PROGRAM main
  VAR
    SYSTEM_ON : BOOL := FALSE;
    SYS_READY : BOOL := FALSE;
    START_MEASURE : BOOL := FALSE;
    PZEM_OK : BOOL := FALSE;
    DATA_READY : BOOL := FALSE;
    MOTOR_ON : BOOL := FALSE;
    STATUS_NORMAL : BOOL := FALSE;
    STATUS_WARNING : BOOL := FALSE;
    STATUS_DANGER : BOOL := FALSE;
    STATUS_OFF : BOOL := FALSE;
    VOLTAGE : REAL := 220.0;
    CURRENT : REAL := 0.138;
    FREQUENCY : REAL := 50.0;
    CAPACITANCE : REAL := 0.00;
    ERROR_PERCENT : REAL := 0.00;
    TIMER_1H : TON;
    READ_PZEM : BOOL := FALSE;
  END_VAR
  VAR  (* added by the conversion: wires and edge detectors of the diagram *)
    _GT25_OUT : BOOL;
  END_VAR

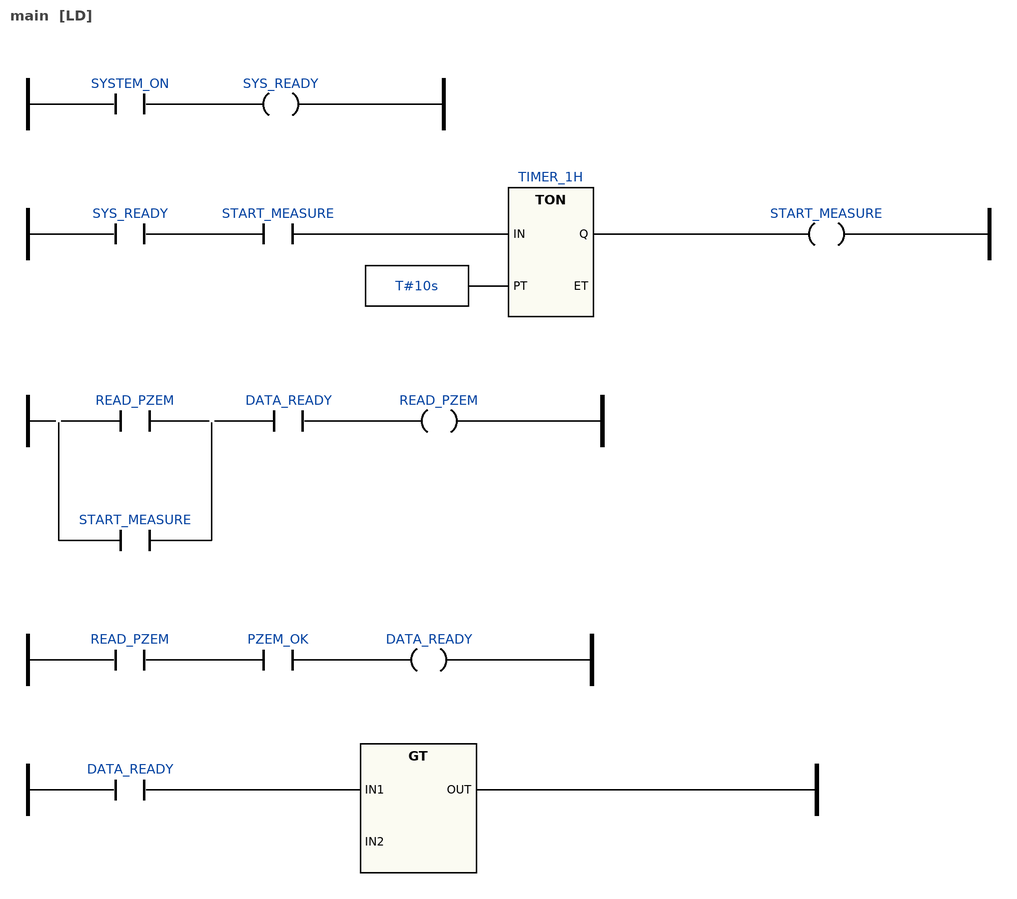
(* LD diagram, written out as Structured Text *)
SYS_READY := SYSTEM_ON;
TIMER_1H(IN := SYS_READY AND START_MEASURE, PT := T#10s);
START_MEASURE := TIMER_1H.Q;
READ_PZEM := (READ_PZEM OR START_MEASURE) AND DATA_READY;
DATA_READY := READ_PZEM AND PZEM_OK;
_GT25_OUT := GT(IN1 := DATA_READY);
END_PROGRAM
